	            ELSE // error not known, user have to act - leave block
	              #statInternal.diagnostics.status := #ERR_DATALOG_OPEN;
	              #statInternal.diagnostics.subfunctionStatus := #instDataLogOpen.STATUS;
	              #statInternal.diagnostics.stateNumber := #FB_STATE_DL_OPEN;
	              #statInternal.errorUserCleared := TRUE;
	            END_IF;
	            // reset instance
	            #instDataLogOpen(REQ := FALSE);
	          END_IF;
	        END_REGION DataLog open

	      #FB_STATE_DL_CREATE:
	        REGION DataLog create
	          #instDataLogCreate(REQ       := TRUE,
	                             RECORDS   := #statDataLogCommands.noOfRecords,
	                             TIMESTAMP := #statDataLogCommands.timestampFormat,
	                             NAME      := #statDataLogCommands.name,
	                             ID        := #statDataLogCommands.id,
	                             HEADER    := #statDataLogCommands.header,
	                             DATA      := #data);

	          // check if creating and opening DL is done successfully - goto write
	          IF #instDataLogCreate.DONE THEN
	            IF (#statDataLogCommands.isLoggingByInterval = TRUE) THEN
	              #statMainState := #FB_STATE_DL_WRITE;
	            ELSE // is logging by trigger
	              #statMainState := #FB_STATE_DL_WAIT_FOR_TRIGGER;
	            END_IF;
	            // reset instance
	            #instDataLogCreate(REQ := FALSE);

	            // check if error occurred
	          ELSIF #instDataLogCreate.ERROR THEN
	            // error not known, user have to act
	            #statInternal.diagnostics.status := #ERR_DATALOG_CREATE;
	            #statInternal.diagnostics.subfunctionStatus := #instDataLogCreate.STATUS;
	            #statInternal.diagnostics.stateNumber := #FB_STATE_DL_OPEN;
	            #statInternal.errorUserCleared := TRUE;
	            // reset instance
	            #instDataLogCreate(REQ := FALSE);
	          END_IF;
	        END_REGION DataLog create

	      #FB_STATE_DL_WAIT_FOR_TRIGGER,
	      #FB_STATE_DL_WAIT_FOR_WRITE_CYCLE:
	        REGION Wait for trigger
	          // reset flags
	          #statLlastEntryReached := FALSE;
	          #statInternal.diagnostics.status := #STATUS_SUBSEQUENT_CALL;

	          IF TRUE // if trigger has a rising edge
	            AND (#triggerLogEntry AND NOT #statDataLogCommands.edgeOnTriggerLogEntry)
	            AND (#statMainState = #FB_STATE_DL_WAIT_FOR_TRIGGER)
	          THEN
	            #statMainState := #FB_STATE_DL_WRITE;

	          ELSIF TRUE // if interval is over
	            AND #instIntervalTimer.Q
	            AND (#statMainState = #FB_STATE_DL_WAIT_FOR_WRITE_CYCLE)
	          THEN
	            #statMainState := #FB_STATE_DL_WRITE;
	          END_IF;
	        END_REGION Wait for trigger

	      #FB_STATE_DL_WRITE:
	        REGION DataLog write
	          #instDataLogWrite(REQ := TRUE,
	                            ID  := #statDataLogCommands.id);

	          // check if datalog is at its last entry
	          IF (#instDataLogWrite.STATUS = #DATALOG_LAST_ENTRY_WRITTEN) THEN
	            // set flag
	            #statLlastEntryReached := TRUE;
	            #statInternal.diagnostics.status := #STATUS_MAX_ENTRIES_REACHED;
	            // increment counter
	            #statNoOfEntries += 1;
	            #statWriteEntryDone := TRUE;

	            // check if datalog should be overwritten or not
	            IF #statDataLogCommands.enableRingBuffer THEN
	              // is logging by interval
	              IF #statDataLogCommands.isLoggingByInterval THEN
	                #statMainState := #FB_STATE_DL_WAIT_FOR_WRITE_CYCLE;

	              ELSE // is logging by trigger
	                #statMainState := #FB_STATE_DL_WAIT_FOR_TRIGGER;
	              END_IF;

	            ELSE // do not overwrite - disable and leave block
	              #statMainState := #FB_STATE_NO_PROCESSING;
	            END_IF;
	            // reset instance
	            #instDataLogWrite(REQ := FALSE);
	            #tempExitStateLoop := FALSE;

	            // check if open DL is done successfully - goto write
	          ELSIF #instDataLogWrite.DONE THEN
	            // increment counter
	            #statNoOfEntries += 1;
	            #statWriteEntryDone := TRUE;

	            IF #statDataLogCommands.isLoggingByInterval = TRUE THEN
	              #statMainState := #FB_STATE_DL_WAIT_FOR_WRITE_CYCLE;
	            ELSE // is logging by trigger
	              #statMainState := #FB_STATE_DL_WAIT_FOR_TRIGGER;
	            END_IF;
	            // reset instance
	            #instDataLogWrite(REQ := FALSE);
	            #tempExitStateLoop := FALSE;

	            // check if error occurred
	          ELSIF #instDataLogWrite.ERROR THEN
	            // error not known, user have to act
	            #statInternal.diagnostics.status := #ERR_DATALOG_WRITE;
	            #statInternal.diagnostics.subfunctionStatus := #instDataLogWrite.STATUS;
	            #statInternal.diagnostics.stateNumber := #FB_STATE_DL_WRITE;
	            #statInternal.errorAutoCleared := TRUE;
	            #statMainState := #FB_STATE_NO_PROCESSING;
	            // reset instance
	            #instDataLogWrite(REQ := FALSE);
	          END_IF;
	        END_REGION DataLog write

	      #FB_STATE_DL_CLEAR:
	        REGION DataLog clear
	          #instDataLogClear(REQ := TRUE,
	                            ID  := #statDataLogCommands.id);

	          // check if open DL is done successfully - goto write
	          IF #instDataLogClear.DONE THEN
	            #statMainState := #FB_STATE_DL_CLEAR_DONE;
	            // reset flag
	            #statLlastEntryReached := FALSE;
	            #statNoOfEntries := 0;
	            // reset instance
	            #instDataLogClear(REQ := FALSE);

	            // check if error occurred
	          ELSIF #instDataLogClear.ERROR THEN
	            // error not known, user have to act
	            #statInternal.diagnostics.status := #ERR_DATALOG_CLEAR;
	            #statInternal.diagnostics.subfunctionStatus := #instDataLogClear.STATUS;
	            #statInternal.diagnostics.stateNumber := #FB_STATE_DL_CLEAR;
	            #statInternal.errorAutoCleared := TRUE;
	            #statMainState := #FB_STATE_NO_PROCESSING;
	            // reset instance
	            #instDataLogWrite(REQ := FALSE);
	          END_IF;
	        END_REGION DataLog clear

	      #FB_STATE_DL_CLEAR_DONE:
	        REGION DataLog clear done
	          IF NOT #clearLog THEN
	            IF #statDataLogCommands.isLoggingByInterval THEN
	              #statMainState := #FB_STATE_DL_WRITE;
	            ELSE
	              #statMainState := #FB_STATE_DL_WAIT_FOR_TRIGGER;
	            END_IF;
	          END_IF;
	        END_REGION DataLog clear

	      #FB_STATE_DL_DELETE:
	        REGION DataLog delete
	          #instDataLogDelete(REQ     := TRUE,
	                             NAME    := #statDataLogCommands.name,
	                             DelFile := #parameter.deleteFile,
	                             ID      := #statDataLogCommands.id);

	          // check if delete DL is done successfully - goto disable completed
	          IF #instDataLogDelete.DONE THEN
	            #statMainState := #FB_STATE_DL_DELETE_DONE;
	            // reset flag
	            #statLlastEntryReached := FALSE;
	            #statNoOfEntries := 0;
	            // reset instance
	            #instDataLogDelete(REQ := FALSE);

	            // check if error occurred
	          ELSIF #instDataLogDelete.ERROR THEN
	            // error not known, user have to act
	            #statInternal.diagnostics.status := #ERR_DATALOG_DELETE;
	            #statInternal.diagnostics.subfunctionStatus := #instDataLogDelete.STATUS;
	            #statInternal.diagnostics.stateNumber := #FB_STATE_DL_DELETE;
	            #statInternal.errorAutoCleared := TRUE;
	            #statMainState := #FB_STATE_NO_PROCESSING;
	            // reset instance
	            #instDataLogDelete(REQ := FALSE);
	          END_IF;
	        END_REGION DataLog delete

	      #FB_STATE_DL_DELETE_DONE:
	        REGION DataLog delete done
	          IF NOT #deleteLog THEN
	            #statMainState := #FB_STATE_DISABLING_COMPLETED;
	          END_IF;
	        END_REGION DataLog delete

	      #FB_STATE_DISABLING: // Disabling active
	        REGION Disabling
	          // closing DataLog
	          #instDataLogClose(REQ := TRUE,
	                            ID  := #statDataLogCommands.id);

	          // check if datalog is closed
	          IF FALSE
	            OR #instDataLogClose.DONE
	            OR #instDataLogClose.STATUS = #SUB_ERR_DATALOG_DOSE_NOT_EXIST
	          THEN
	            #statMainState := #FB_STATE_DISABLING_COMPLETED;
	            #statInternal.diagnostics.status := #STATUS_FINISHED_NO_ERROR;

	            // if closing ends with error - report this as well
	          ELSIF #instDataLogClose.ERROR THEN
	            // error occurred - copy to outputs
	            #statInternal.diagnostics.status := #ERR_DATALOG_CLOSE;
	            #statInternal.diagnostics.subfunctionStatus := #instDataLogClose.STATUS;
	            #statInternal.diagnostics.stateNumber := #FB_STATE_DISABLING;
	            #statInternal.errorAutoCleared := TRUE;// next state
	            #statMainState := #FB_STATE_DISABLING_COMPLETED;
	          END_IF;
	        END_REGION Disabling

	      #FB_STATE_DISABLING_COMPLETED:
	        REGION Disabling completed
	          // reset instance
	          #instDataLogClose(REQ := FALSE);
	          // When disabling is complete the bit #statDisablingCompleted must be set
	          #statInternal.disablingCompleted := TRUE;
	        END_REGION Disabling completed

	      ELSE // Undefined state in state machine reached
	        REGION Undefined state
	          #statInternal.diagnostics.status := #ERR_UNDEFINED_STATE;
	          #statInternal.diagnostics.subfunctionStatus := #SUB_STATUS_NO_ERROR;
	          #statInternal.diagnostics.stateNumber := #statMainState;
	          #statInternal.errorUserCleared := TRUE;
	        END_REGION Undefined state
	    END_CASE;

	    // call interval timer
	    #instIntervalTimer.TON(IN := (#statMainState = #FB_STATE_DL_WAIT_FOR_WRITE_CYCLE),
	                           PT := #statDataLogCommands.loggingInterval);    // if one ore more runs in the same cycle are necessary, set #tempExitStateLoop := FALSE;
	    // check state, if condition = TRUE --> #tempExitStateLoop = TRUE --> LEAVE LOOP
	  UNTIL (TRUE = #tempExitStateLoop)
	  END_REPEAT;
	END_REGION STATE_MACHINE

	REGION Edge memory
	  // store/ reset edge memory
	  #statDataLogCommands.edgeOnTriggerLogEntry := #triggerLogEntry;
	  #statDataLogCommands.clearLogPrevious := #clearLog;
	  #statDataLogCommands.deleteLogPrevious := #deleteLog;
	END_REGION

	REGION OUTPUTS
	  // Write outputs
	  IF (#statInternal.disablingCompleted = TRUE) THEN
	    REGION disabling
	      // Reset outputs if disabling completed
	      #statInternal.valid := FALSE;
	      #statInternal.busy := FALSE;
	      #statInternal.error := FALSE;
	      #statInternal.errorUserCleared := FALSE;
	      #statInternal.errorAutoCleared := FALSE;
	      #statInternal.diagnostics.status := #STATUS_NO_CALL;
	      // Reset application specific outputs
	      #statWriteEntryDone := FALSE;
	    END_REGION disabling

	  ELSIF (#statInternal.errorUserCleared = TRUE) AND (#statInternal.error = FALSE) THEN
	    REGION error user cleared
	      // Error can only be cleared by user; rising edge at enable input is needed to continue
	      #statInternal.valid := FALSE;
	      #statInternal.busy := FALSE;
	      #statInternal.error := TRUE;
	      // Write diagnostics
	      #diagnostics := #statInternal.diagnostics;
	      // Reset application specific outputs
	      #statWriteEntryDone := FALSE;
	      // execution aborted --> set state no processing
	      #statMainState := #FB_STATE_NO_PROCESSING;
	    END_REGION error user cleared

	  ELSIF (#statInternal.errorAutoCleared = TRUE) AND (#statInternal.error = FALSE) THEN
	    REGION error auto cleared
	      // Error can be reset by FB automatically
	      #statInternal.valid := FALSE;
	      #statInternal.busy := TRUE;
	      #statInternal.error := TRUE;
	      // Write diagnostics
	      #diagnostics := #statInternal.diagnostics;
	      // Reset application specific outputs
	      #statWriteEntryDone := FALSE;
	    END_REGION error auto cleared

	  ELSIF (#statInternal.errorAutoCleared = FALSE) AND (#statInternal.errorUserCleared = FALSE) AND (#statInternal.error = TRUE) THEN
	    REGION after user/auto cleared
	      // If autocleared error is acknowledged
	      #statInternal.valid := TRUE;
	      #statInternal.busy := TRUE;
	      #statInternal.error := FALSE;
	      // remove this line if more detailed status information is used instead of "#STATUS_SUBSEQUENT_CALL"
	      #statInternal.diagnostics.status := #STATUS_SUBSEQUENT_CALL;
	    END_REGION after user/auto cleared
	  END_IF;

	  REGION Write static values to outputs
	    #valid := #statInternal.valid;
	    #busy := #statInternal.busy;
	    #error := #statInternal.error;
	    #status := #statInternal.diagnostics.status;
	    // if ENO mechanism is not used / not wanted replace the following line by --> ENO := TRUE;
	    ENO := NOT #statInternal.error;
	    // Write application specific static values to outputs
	    #lastEntryReached := #statLlastEntryReached;
	    #noOfEntries := #statNoOfEntries;

	    #writeEntryDone := #statWriteEntryDone;
	    #statWriteEntryDone := FALSE;

	    #clearLogDone := #statMainState = #FB_STATE_DL_CLEAR_DONE;
	    #deleteLogDone := #statMainState = #FB_STATE_DL_DELETE_DONE;
	  END_REGION Write static values to outputs
	END_REGION OUTPUTS

END_FUNCTION_BLOCK

FUNCTION "LGF_IsParityOdd" : Bool
{ S7_Optimized_Access := 'TRUE' }
AUTHOR : Siemens_SIMATIC_Systems_Support
FAMILY : LGF
NAME : LGF_IsParityOdd
   VAR_INPUT
      doubleWord : DWord;
   END_VAR

   VAR_TEMP
      tempDword : DWord;
   END_VAR

   VAR CONSTANT
      SHIFT_ONE_BIT : USInt := 1;
      SHIFT_TWO_BIT : USInt := 2;
      SHIFT_TO_RESULT : USInt := 28;
      MASK_FOR_RESULT : DWord := 16#11111111;
   END_VAR


BEGIN
	REGION Block info header
	  //============================================================================
	  // SIEMENS AG / (c)Copyright 2018
	  //----------------------------------------------------------------------------
	  // Title:            LGF_IsParityOdd
	  // Comment/Function: check if parity in input tag is odd
	  //                   if number of bits is odd, return TRUE
	  //                   https://graphics.stanford.edu/~seander/bithacks.html#ParityMultiply
	  //                   ENO not needed, no error possible
	  // Library/Family:   LGF (Library General Functions)
	  // Author:           Siemens Digital Industry Support
	  // Tested with:      S7-PLCSIM Advanced V2.0 SP1
	  // Engineering:      TIA Portal V15 Update 2
	  // Restrictions:     ENO not needed, no error possible
	  // Requirements:     PLC (S7-1200 / S7-1500)
	  //-------------------------------------------------------------------------------
	  // Change log table:
	  // Version  | Date       | Expert in charge       | Changes applied
	  //----------|------------|------------------------|------------------------------
	  // 01.00.00 | 2019.11.28 | Simatic Systems Support
	  //                         First released version
	  // 03.00.00 | 23.04.2020 | Simatic Systems Support | Set version to V3.0.0
	  //                         harmonize the version of the whole library
	  // 03.00.01 | 12.11.2020 | Simatic Systems Support
	  //                         Insert documentation
	  //=============================================================================
	END_REGION Block info header

	REGION DESCRIPTION
	  (/**/)
	END_REGION DESCRIPTION

	REGION Logic
	  #tempDword := #doubleWord; // 32-bit word
	  #tempDword := #tempDword XOR SHR(IN := #tempDword, N := #SHIFT_ONE_BIT);
	  #tempDword := #tempDword XOR SHR(IN := #tempDword, N := #SHIFT_TWO_BIT);

	  #tempDword := UDINT_TO_DWORD(DWORD_TO_UDINT(#tempDword AND #MASK_FOR_RESULT) * DWORD_TO_UDINT(#MASK_FOR_RESULT));

	  #tempDword := SHR(IN := #tempDword, N := #SHIFT_TO_RESULT);

	  // result is stored in LSB
	  #LGF_IsParityOdd := #tempDword.%X0;

	  // eno not needed, no error possible
	  ENO := FALSE;
	END_REGION

END_FUNCTION

FUNCTION "LGF_CalcCRC32Advanced" : DWord
{ S7_Optimized_Access := 'TRUE' }
AUTHOR : Siemens_Industry_Support
FAMILY : LGF
NAME : LGF_CRC32Advanced
   VAR_INPUT
      initValue { S7_PredefinedAssignment := '16#00'} : DWord;
      mask { S7_PredefinedAssignment := '16#00'} : DWord;
      finalXorValue { S7_PredefinedAssignment := '16#00'} : DWord;
      reflectInput { S7_PredefinedAssignment := 'FALSE'} : Bool;
      reflectResult { S7_PredefinedAssignment := 'FALSE'} : Bool;
      noOfElements { S7_PredefinedAssignment := '0'} : UInt;
   END_VAR

   VAR_OUTPUT
      error : Bool;
      status : Word;
   END_VAR

   VAR_IN_OUT
      "array" : Array[*] of Byte;
   END_VAR

   VAR_TEMP
      tempInput : Byte;
      tempCRC : DWord;
      tempInvCRC : DWord;
      tempLowerLimit : DInt;
      tempUpperLimit : DInt;
      tempIndexArray : DInt;
      tempIndexCRC : DInt;
   END_VAR

   VAR CONSTANT
      SHIFT_ONE_BIT : UInt := 1;
      SHIFT_THREE_BYTE : UInt := 24;
      ARRAY_FIRST_DIMENSION : UInt := 1;
      CRC_LOOP_LOWER_LIMIT : DInt := 0;
      CRC_LOOP_UPPER_LIMIT : DInt := 7;
      STATUS_NO_ERROR : Word := 16#0000;
      ERR_NO_OF_ELEMENTS : Word := 16#8400;
   END_VAR


BEGIN
	REGION Block info header
	  //===============================================================================
	  // SIEMENS AG / (c)Copyright 2019
	  //-------------------------------------------------------------------------------
	  // Title:            LGF_CRC32Advanced
	  // Comment/Function: This function makes a CRC calculation according
	  //                   to the CRC-32 algorithm
	  //                   advanced because of reflect In/Out and final XOR combination
	  // Library/Family:   LGF (Library General Functions)
	  // Author:           Siemens Digital Industry Support
	  // Tested with:      CPU 1515F-2 PN FW:V2.6
	  // Engineering:      TIA Portal V15.1 Update 2
	  // Restrictions:     ENO disabled - no error handling, no failure possible
	  // Requirements:     PLC (S7-1200 / S7-1500)
	  //-------------------------------------------------------------------------------
	  // Change log table:
	  // Version  | Date       | Expert in charge       | Changes applied
	  //----------|------------|------------------------|------------------------------
	  // 01.00.00 03.07.2018  Siemens Industry Online Support
	  //                      First released version
	  // 01.00.01 17.08.2018  Siemens Industry Online Support
	  //                      Upgrade: TIA V15 Update 2
	  // 01.00.02 23.11.2018  Siemens Industry Online Support
	  //                      Upgrade: TIA V15.1
	  // 01.00.03 09.10.2019  Simatic Systems Support
	  //                      Code refactoring, comments added
	  // 03.00.00 23.04.2020  Simatic Systems Support
	  //                      Set version to V3.0.0, harmonize the version of the whole library
	  // 03.00.01 12.11.2020  Simatic Systems Support
	  //                      Insert documentation
	  //                      Assign default start values to optional inputs - `initValue`, `mask`, `finalXorValue`, `reflectInput`, `reflectResult`
	  // 03.01.00 14.04.2023  Simatic Systems Support
	  //                      Add input `noOfElements` to assign length to be converted different from array size
	  //                      Add outputs `error` and `status` display a wrong assignment to `noOfElements`
	  //=============================================================================
	END_REGION Block info header

	REGION DESCRIPTION
	  (/**/)
	END_REGION DESCRIPTION

	REGION Initialization and input data processing
	  // Defining initial value for algorithm
	  #tempCRC := #initValue;
	  // Input array size calculation
	  #tempLowerLimit := LOWER_BOUND(ARR := #array, DIM := #ARRAY_FIRST_DIMENSION);
	  #tempUpperLimit := UPPER_BOUND(ARR := #array, DIM := #ARRAY_FIRST_DIMENSION);

	  // check paramter `noOfELements`, if gretaer than zero check if fits to array size
	  IF #noOfElements > 0 THEN
	    IF #noOfElements > (#tempUpperLimit - #tempLowerLimit + 1) THEN
	      #status := #ERR_NO_OF_ELEMENTS;
	      #error := TRUE;
	      ENO := FALSE;
	      #LGF_CalcCRC32Advanced := #tempCRC;
	      RETURN;
	    ELSE
	      #tempUpperLimit := #tempLowerLimit + #noOfElements - 1;
	    END_IF;
	  END_IF;
	END_REGION

	REGION CRC calculation
	  FOR #tempIndexArray := #tempLowerLimit TO #tempUpperLimit DO

	    IF #reflectInput THEN
	      // Reverse bit order in input byte
	      #tempInput.%X7 := #array[#tempIndexArray].%X0;
	      #tempInput.%X6 := #array[#tempIndexArray].%X1;
	      #tempInput.%X5 := #array[#tempIndexArray].%X2;
	      #tempInput.%X4 := #array[#tempIndexArray].%X3;
	      #tempInput.%X3 := #array[#tempIndexArray].%X4;
	      #tempInput.%X2 := #array[#tempIndexArray].%X5;
	      #tempInput.%X1 := #array[#tempIndexArray].%X6;
	      #tempInput.%X0 := #array[#tempIndexArray].%X7;
	    ELSE
	      #tempInput := #array[#tempIndexArray];
	    END_IF;

	    // Perform division using XOR function for appropriate DWord in array (with shift byte into MSB of 32bit CRC)
	    #tempCRC := #tempCRC XOR SHL(IN := BYTE_TO_DWORD(#tempInput), N := #SHIFT_THREE_BYTE);

	    FOR #tempIndexCRC := #CRC_LOOP_LOWER_LIMIT TO #CRC_LOOP_UPPER_LIMIT DO
	      // Check if MSB is set
	      IF #tempCRC.%X31 THEN
	        // Shift left and perform division by mask polynomial using XOR function
	        #tempCRC := SHL(IN := #tempCRC, N := #SHIFT_ONE_BIT) XOR #mask;
	      ELSE
	        // Shift left without division
	        #tempCRC := SHL(IN := #tempCRC, N := #SHIFT_ONE_BIT);
	      END_IF;
	    END_FOR;

	  END_FOR;
	END_REGION

	REGION Outputs assignment
	  IF #reflectResult THEN
	    // Reverse bit order in CRC checksum
	    #tempInvCRC.%X31 := #tempCRC.%X0;
	    #tempInvCRC.%X30 := #tempCRC.%X1;
	    #tempInvCRC.%X29 := #tempCRC.%X2;
	    #tempInvCRC.%X28 := #tempCRC.%X3;
	    #tempInvCRC.%X27 := #tempCRC.%X4;
	    #tempInvCRC.%X26 := #tempCRC.%X5;
	    #tempInvCRC.%X25 := #tempCRC.%X6;
	    #tempInvCRC.%X24 := #tempCRC.%X7;
	    #tempInvCRC.%X23 := #tempCRC.%X8;
	    #tempInvCRC.%X22 := #tempCRC.%X9;
	    #tempInvCRC.%X21 := #tempCRC.%X10;
	    #tempInvCRC.%X20 := #tempCRC.%X11;
	    #tempInvCRC.%X19 := #tempCRC.%X12;
	    #tempInvCRC.%X18 := #tempCRC.%X13;
	    #tempInvCRC.%X17 := #tempCRC.%X14;
	    #tempInvCRC.%X16 := #tempCRC.%X15;
	    #tempInvCRC.%X15 := #tempCRC.%X16;
	    #tempInvCRC.%X14 := #tempCRC.%X17;
	    #tempInvCRC.%X13 := #tempCRC.%X18;
	    #tempInvCRC.%X12 := #tempCRC.%X19;
	    #tempInvCRC.%X11 := #tempCRC.%X20;
	    #tempInvCRC.%X10 := #tempCRC.%X21;
	    #tempInvCRC.%X9 := #tempCRC.%X22;
	    #tempInvCRC.%X8 := #tempCRC.%X23;
	    #tempInvCRC.%X7 := #tempCRC.%X24;
	    #tempInvCRC.%X6 := #tempCRC.%X25;
	    #tempInvCRC.%X5 := #tempCRC.%X26;
	    #tempInvCRC.%X4 := #tempCRC.%X27;
	    #tempInvCRC.%X3 := #tempCRC.%X28;
	    #tempInvCRC.%X2 := #tempCRC.%X29;
	    #tempInvCRC.%X1 := #tempCRC.%X30;
	    #tempInvCRC.%X0 := #tempCRC.%X31;

	    #LGF_CalcCRC32Advanced := #tempInvCRC XOR #finalXorValue;
	  ELSE
	    #LGF_CalcCRC32Advanced := #tempCRC XOR #finalXorValue;
	  END_IF;

	  #status := #STATUS_NO_ERROR;
	  #error := FALSE;
	  ENO := TRUE;
	END_REGION

END_FUNCTION

FUNCTION "LGF_CalcCRC32" : DWord
{ S7_Optimized_Access := 'TRUE' }
AUTHOR : Siemens_Industry_Support
FAMILY : LGF
NAME : LGF_CRC32
   VAR_INPUT
      initValue { S7_PredefinedAssignment := '16#00'} : DWord;
      mask { S7_PredefinedAssignment := '16#00'} : DWord;
      noOfElements { S7_PredefinedAssignment := '0'} : UInt;
   END_VAR

   VAR_OUTPUT
      error : Bool;
      status : Word;
   END_VAR

   VAR_IN_OUT
      "array" : Array[*] of Byte;
   END_VAR

   VAR_TEMP
      tempCRC : DWord;
      tempLowerLimit : DInt;
      tempUpperLimit : DInt;
      tempIndexArray : DInt;
      tempIndexCRC : DInt;
   END_VAR

   VAR CONSTANT
      SHIFT_ONE_BIT : UInt := 1;
      SHIFT_THREE_BYTES : UInt := 24;
      ARRAY_FIRST_DIMENSION : UInt := 1;
      CRC_LOOP_LOWER_LIMIT : DInt := 0;
      CRC_LOOP_UPPER_LIMIT : DInt := 7;
      STATUS_NO_ERROR : Word := 16#0000;
      ERR_NO_OF_ELEMENTS : Word := 16#8400;
   END_VAR


BEGIN
	REGION Block info header
	  //===============================================================================
	  // SIEMENS AG / (c)Copyright 2019
	  //-------------------------------------------------------------------------------
	  // Title:            LGF_CRC32
	  // Comment/Function: This function makes a CRC calculation according
	  //                   to the CRC-32 algorithm
	  // Library/Family:   LGF (Library General Functions)
	  // Author:           Siemens Digital Industry Support
	  // Tested with:      CPU 1515F-2 PN FW:V2.6
	  // Engineering:      TIA Portal V15.1 Update 2
	  // Restrictions:     ENO disabled - no error handling, no failure possible
	  // Requirements:     PLC (S7-1200 / S7-1500)
	  //-------------------------------------------------------------------------------
	  // Change log table:
	  // Version  | Date       | Expert in charge       | Changes applied
	  //----------|------------|------------------------|------------------------------
	  // 01.00.00 03.07.2018  Siemens Industry Online Support
	  //                      First released version
	  // 01.00.01 17.08.2018  Siemens Industry Online Support
	  //                      Upgrade: TIA V15 Update 2
	  // 01.00.02 23.11.2018  Siemens Industry Online Support
	  //                      Upgrade: TIA V15.1
	  // 01.00.03 09.10.2019  Simatic Systems Support
	  //                      Code refactoring, comments added
	  // 03.00.00 23.04.2020  Simatic Systems Support
	  //                      Set version to V3.0.0, harmonize the version of the whole library
	  // 03.00.01 12.11.2020  Simatic Systems Support
	  //                      Insert documentation
	  //                      Assign default start values to optional inputs - `initValue`, `mask`
	  // 03.01.00 14.04.2023  Simatic Systems Support
	  //                      Add input `noOfElements` to assign length to be converted different from array size
	  //                      Add outputs `error` and `status` display a wrong assignment to `noOfElements`
	  //=============================================================================
	END_REGION Block info header

	REGION DESCRIPTION
	  (/**/)
	END_REGION DESCRIPTION

	REGION Initialization and input data processing
	  // Defining initial value for algorithm
	  #tempCRC := #initValue;
	  // Input array size calculation
	  #tempLowerLimit := LOWER_BOUND(ARR := #array, DIM := #ARRAY_FIRST_DIMENSION);
	  #tempUpperLimit := UPPER_BOUND(ARR := #array, DIM := #ARRAY_FIRST_DIMENSION);

	  // check paramter `noOfELements`, if gretaer than zero check if fits to array size
	  IF #noOfElements > 0 THEN
	    IF #noOfElements > (#tempUpperLimit - #tempLowerLimit + 1) THEN
	      #status := #ERR_NO_OF_ELEMENTS;
	      #error := TRUE;
	      ENO := FALSE;
	      #LGF_CalcCRC32 := #tempCRC;
	      RETURN;
	    ELSE
	      #tempUpperLimit := #tempLowerLimit + #noOfElements - 1;
	    END_IF;
	  END_IF;
	END_REGION

	REGION CRC calculation
	  FOR #tempIndexArray := #tempLowerLimit TO #tempUpperLimit DO
	    // Perform division using XOR function for appropriate word in array (with shift byte into MSB of 32bit CRC)
	    #tempCRC := #tempCRC XOR SHL(IN := BYTE_TO_DWORD(#array[#tempIndexArray]), N := #SHIFT_THREE_BYTES);

	    FOR #tempIndexCRC := #CRC_LOOP_LOWER_LIMIT TO #CRC_LOOP_UPPER_LIMIT DO
	      // Check if MSB is set
	      IF #tempCRC.%X31 THEN
	        // Shift left and perform division by mask polynomial using XOR function
	        #tempCRC := SHL(IN := #tempCRC, N := #SHIFT_ONE_BIT) XOR #mask;
	      ELSE
	        // Shift left without division
	        #tempCRC := SHL(IN := #tempCRC, N := #SHIFT_ONE_BIT);
	      END_IF;
	    END_FOR;

	  END_FOR;
	END_REGION

	REGION Outputs assignment
	  #LGF_CalcCRC32 := #tempCRC;

	  #status := #STATUS_NO_ERROR;
	  #error := FALSE;
	  ENO := TRUE;
	END_REGION

END_FUNCTION

FUNCTION "LGF_CalcCRC16Advanced" : Word
{ S7_Optimized_Access := 'TRUE' }
AUTHOR : Siemens_Industry_Support
FAMILY : LGF
NAME : LGF_CRC16Advanced
   VAR_INPUT
      initValue { S7_PredefinedAssignment := '16#00'} : Word;
      mask { S7_PredefinedAssignment := '16#00'} : Word;
      finalXorValue { S7_PredefinedAssignment := '16#00'} : Word;
      reflectInput { S7_PredefinedAssignment := 'FALSE'} : Bool;
      reflectResult { S7_PredefinedAssignment := 'FALSE'} : Bool;
      noOfElements { S7_PredefinedAssignment := '0'} : UInt;
   END_VAR

   VAR_OUTPUT
      error : Bool;
      status : Word;
   END_VAR

   VAR_IN_OUT
      "array" : Array[*] of Byte;
   END_VAR

   VAR_TEMP
      tempInput : Byte;
      tempCRC : Word;
      tempInvCRC : Word;
      tempLowerLimit : DInt;
      tempUpperLimit : DInt;
      tempIndexArray : DInt;
      tempIndexCRC : DInt;
   END_VAR

   VAR CONSTANT
      SHIFT_ONE_BIT : UInt := 1;
      SHIFT_ONE_BYTE : UInt := 8;
      ARRAY_FIRST_DIMENSION : UInt := 1;
      CRC_LOOP_LOWER_LIMIT : DInt := 0;
      CRC_LOOP_UPPER_LIMIT : DInt := 7;
      STATUS_NO_ERROR : Word := 16#0000;
      ERR_NO_OF_ELEMENTS : Word := 16#8400;
   END_VAR


BEGIN
	REGION Block info header
	  //===============================================================================
	  // SIEMENS AG / (c)Copyright 2019
	  //-------------------------------------------------------------------------------
	  // Title:            LGF_CRC16Advanced
	  // Comment/Function: This function makes a CRC calculation according
	  //                   to the CRC-16 advanced algorithm
	  //                   advanced because of reflect In/Out and final XOR combination
	  // Library/Family:   LGF (Library General Functions)
	  // Author:           Siemens Digital Industry Support
	  // Tested with:      CPU 1515F-2 PN FW:V2.6
	  // Engineering:      TIA Portal V15.1 Update 2
	  // Restrictions:     ENO disabled - no error handling, no failure possible
	  // Requirements:     PLC (S7-1200 / S7-1500)
	  //-------------------------------------------------------------------------------
	  // Change log table:
	  // Version  | Date       | Expert in charge       | Changes applied
	  //----------|------------|------------------------|------------------------------
	  // 01.00.00 16.12.2019  Simatic Systems Support
	  //                      first release, copied from "LGF_CalcCRC32Advanced"
	  // 03.00.00 23.04.2020  Simatic Systems Support
	  //                      Set version to V3.0.0, harmonize the version of the whole library
	  // 03.00.01 12.11.2020  Simatic Systems Support
	  //                      Insert documentation
	  //                      Assign default start values to optional inputs - `initValue`, `mask`, `finalXorValue`, `reflectInput`, `reflectResult`
	  // 03.01.00 14.04.2023  Simatic Systems Support
	  //                      Add input `noOfElements` to assign length to be converted different from array size
	  //                      Add outputs `error` and `status` display a wrong assignment to `noOfElements`
	  //=============================================================================
	END_REGION Block info header

	REGION DESCRIPTION
	  (/**/)
	END_REGION DESCRIPTION

	REGION Initialization and input data processing
	  // Defining initial value for algorithm
	  #tempCRC := #initValue;
	  // Input array size calculation
	  #tempLowerLimit := LOWER_BOUND(ARR := #array, DIM := #ARRAY_FIRST_DIMENSION);
	  #tempUpperLimit := UPPER_BOUND(ARR := #array, DIM := #ARRAY_FIRST_DIMENSION);

	  // check paramter `noOfELements`, if gretaer than zero check if fits to array size
	  IF #noOfElements > 0 THEN
	    IF #noOfElements > (#tempUpperLimit - #tempLowerLimit + 1) THEN
	      #status := #ERR_NO_OF_ELEMENTS;
	      #error := TRUE;
	      ENO := FALSE;
	      #LGF_CalcCRC16Advanced := #tempCRC;
	      RETURN;
	    ELSE
	      #tempUpperLimit := #tempLowerLimit + #noOfElements - 1;
	    END_IF;
	  END_IF;
	END_REGION

	REGION CRC calculation
	  FOR #tempIndexArray := #tempLowerLimit TO #tempUpperLimit DO

	    IF #reflectInput THEN
	      // Reverse bit order in input byte
	      #tempInput.%X7 := #array[#tempIndexArray].%X0;
	      #tempInput.%X6 := #array[#tempIndexArray].%X1;
	      #tempInput.%X5 := #array[#tempIndexArray].%X2;
	      #tempInput.%X4 := #array[#tempIndexArray].%X3;
	      #tempInput.%X3 := #array[#tempIndexArray].%X4;
	      #tempInput.%X2 := #array[#tempIndexArray].%X5;
	      #tempInput.%X1 := #array[#tempIndexArray].%X6;
	      #tempInput.%X0 := #array[#tempIndexArray].%X7;
	    ELSE
	      #tempInput := #array[#tempIndexArray];
	    END_IF;

	    // Perform division using XOR function for appropriate Word in array (with shift byte into MSB of 16bit CRC)
	    #tempCRC := #tempCRC XOR SHL(IN := BYTE_TO_WORD(#tempInput), N := #SHIFT_ONE_BYTE);

	    FOR #tempIndexCRC := #CRC_LOOP_LOWER_LIMIT TO #CRC_LOOP_UPPER_LIMIT DO
	      // Check if MSB is set
	      IF #tempCRC.%X15 THEN
	        // Shift left and perform division by mask polynomial using XOR function
	        #tempCRC := SHL(IN := #tempCRC, N := #SHIFT_ONE_BIT) XOR #mask;
	      ELSE
	        // Shift left without division
	        #tempCRC := SHL(IN := #tempCRC, N := #SHIFT_ONE_BIT);
	      END_IF;
	    END_FOR;

	  END_FOR;
	END_REGION

	REGION Outputs assignment
	  IF #reflectResult THEN
	    // Reverse bit order in CRC checksum
	    #tempInvCRC.%X15 := #tempCRC.%X0;
	    #tempInvCRC.%X14 := #tempCRC.%X1;
	    #tempInvCRC.%X13 := #tempCRC.%X2;
	    #tempInvCRC.%X12 := #tempCRC.%X3;
	    #tempInvCRC.%X11 := #tempCRC.%X4;
	    #tempInvCRC.%X10 := #tempCRC.%X5;
	    #tempInvCRC.%X9 := #tempCRC.%X6;
	    #tempInvCRC.%X8 := #tempCRC.%X7;
	    #tempInvCRC.%X7 := #tempCRC.%X8;
	    #tempInvCRC.%X6 := #tempCRC.%X9;
	    #tempInvCRC.%X5 := #tempCRC.%X10;
	    #tempInvCRC.%X4 := #tempCRC.%X11;
	    #tempInvCRC.%X3 := #tempCRC.%X12;
	    #tempInvCRC.%X2 := #tempCRC.%X13;
	    #tempInvCRC.%X1 := #tempCRC.%X14;
	    #tempInvCRC.%X0 := #tempCRC.%X15;

	    #LGF_CalcCRC16Advanced := #tempInvCRC XOR #finalXorValue;
	  ELSE
	    #LGF_CalcCRC16Advanced := #tempCRC XOR #finalXorValue;
	  END_IF;

	  #status := #STATUS_NO_ERROR;
	  #error := FALSE;
	  ENO := TRUE;
	END_REGION

END_FUNCTION

FUNCTION "LGF_CalcCRC16" : Word
{ S7_Optimized_Access := 'TRUE' }
AUTHOR : Siemens_Industry_Support
FAMILY : LGF
NAME : LGF_CRC16
   VAR_INPUT
      initValue { S7_PredefinedAssignment := '16#00'} : Word;
      mask { S7_PredefinedAssignment := '16#00'} : Word;
      noOfElements { S7_PredefinedAssignment := '0'} : UInt;
   END_VAR

   VAR_OUTPUT
      error : Bool;
      status : Word;
   END_VAR

   VAR_IN_OUT
      "array" : Array[*] of Byte;
   END_VAR

   VAR_TEMP
      tempCRC : Word;
      tempLowerLimit : DInt;
      tempUpperLimit : DInt;
      tempIndexArray : DInt;
      tempIndexCRC : DInt;
   END_VAR

   VAR CONSTANT
      SHIFT_ONE_BIT : UInt := 1;
      SHIFT_ONE_BYTE : UInt := 8;
      ARRAY_FIRST_DIMENSION : UInt := 1;
      CRC_LOOP_LOWER_LIMIT : DInt := 0;
      CRC_LOOP_UPPER_LIMIT : DInt := 7;
      ERR_NO_OF_ELEMENTS : Word := 16#8400;
      STATUS_NO_ERROR : Word := 16#0000;
   END_VAR


BEGIN
	REGION Block info header
	  //===============================================================================
	  // SIEMENS AG / (c)Copyright 2019
	  //-------------------------------------------------------------------------------
	  // Title:            LGF_CRC16
	  // Comment/Function: This function makes a CRC calculation according
	  //                   to the CRC-16 algorithm
	  // Library/Family:   LGF (Library General Functions)
	  // Author:           Siemens Digital Industry Support
	  // Tested with:      CPU 1515F-2 PN FW:V2.6
	  // Engineering:      TIA Portal V15.1 Update 2
	  // Restrictions:     ENO disabled - no error handling, no failure possible
	  // Requirements:     PLC (S7-1200 / S7-1500)
	  //-------------------------------------------------------------------------------
	  // Change log table:
	  // Version  | Date       | Expert in charge       | Changes applied
	  //----------|------------|------------------------|------------------------------
	  // 01.00.00 03.07.2018  Siemens Industry Online Support
	  //                      First released version
	  // 01.00.01 17.08.2018  Siemens Industry Online Support
	  //                      Upgrade: TIA V15 Update 2
	  // 01.00.02 23.11.2018  Siemens Industry Online Support
	  //                      Upgrade: TIA V15.1
	  // 01.00.03 09.10.2019  Simatic Systems Support
	  //                      Code refactoring, comments added
	  // 03.00.00 23.04.2020  Simatic Systems Support
	  //                      Set version to V3.0.0, harmonize the version of the whole library
	  // 03.00.01 12.11.2020  Simatic Systems Support
	  //                      Insert documentation
	  //                      Assign default start values to optional inputs - `initValue`, `mask`
	  // 03.01.00 14.04.2023  Simatic Systems Support
	  //                      Add input `noOfElements` to assign length to be converted different from array size
	  //                      Add outputs `error` and `status` display a wrong assignment to `noOfElements`
	  //=============================================================================
	END_REGION Block info header

	REGION DESCRIPTION
	  (/**/)
	END_REGION DESCRIPTION

	REGION Initialization and input data processing
	  // Defining initial value for algorithm
	  #tempCRC := #initValue;
	  // Input array size calculation
	  #tempLowerLimit := LOWER_BOUND(ARR := #array, DIM := #ARRAY_FIRST_DIMENSION);
	  #tempUpperLimit := UPPER_BOUND(ARR := #array, DIM := #ARRAY_FIRST_DIMENSION);

	  // check paramter `noOfELements`, if gretaer than zero check if fits to array size
	  IF #noOfElements > 0 THEN
	    IF #noOfElements > (#tempUpperLimit - #tempLowerLimit + 1) THEN
	      #status := #ERR_NO_OF_ELEMENTS;
	      #error := TRUE;
	      ENO := FALSE;
	      #LGF_CalcCRC16 := #tempCRC;
	      RETURN;
	    ELSE
	      #tempUpperLimit := #tempLowerLimit + #noOfElements - 1;
	    END_IF;
	  END_IF;
	END_REGION

	REGION CRC calculation
	  FOR #tempIndexArray := #tempLowerLimit TO #tempUpperLimit DO
	    // Perform division using XOR function for appropriate word in array (with shift byte into MSB of 16bit CRC)
	    #tempCRC := #tempCRC XOR SHL(IN := BYTE_TO_WORD(#array[#tempIndexArray]), N := #SHIFT_ONE_BYTE);

	    FOR #tempIndexCRC := #CRC_LOOP_LOWER_LIMIT TO #CRC_LOOP_UPPER_LIMIT DO
	      // Check if MSB is set
	      IF #tempCRC.%X15 THEN
	        // Shift left and perform division by mask polynomial using XOR function
	        #tempCRC := SHL(IN := #tempCRC, N := #SHIFT_ONE_BIT) XOR #mask;
	      ELSE
	        // Shift left without division
	        #tempCRC := SHL(IN := #tempCRC, N := #SHIFT_ONE_BIT);
	      END_IF;
	    END_FOR;

	  END_FOR;
	END_REGION

	REGION Outputs assignment
	  #LGF_CalcCRC16 := #tempCRC;

	  #status := #STATUS_NO_ERROR;
	  #error := FALSE;
	  ENO := TRUE;
	END_REGION

END_FUNCTION

FUNCTION "LGF_CalcCRC8For1Byte" : Byte
{ S7_Optimized_Access := 'TRUE' }
AUTHOR : Siemens_Industry_Support
FAMILY : LGF
NAME : LGF_CRC8For1Byte
   VAR_INPUT
      initValue { S7_PredefinedAssignment := '16#00'} : Byte;
      mask { S7_PredefinedAssignment := '16#00'} : Byte;
      value : Byte;
   END_VAR

   VAR_TEMP
      tempCRC : Byte;
      tempIndexCRC : DInt;
   END_VAR

   VAR CONSTANT
      SHIFT_ONE_BIT : UInt := 1;
      CRC_LOOP_LOWER_LIMIT : DInt := 0;
      CRC_LOOP_UPPER_LIMIT : DInt := 7;
   END_VAR


BEGIN
	REGION Block info header
	  //===============================================================================
	  // SIEMENS AG / (c)Copyright 2019
	  //-------------------------------------------------------------------------------
	  // Title:            LGF_CRC8For1Byte
	  // Comment/Function: This function makes a CRC calculation according
	  //                   to the CRC-8 algorithm for 1 byte
	  // Library/Family:   LGF (Library General Functions)
	  // Author:           Siemens Digital Industry Support
	  // Tested with:      CPU 1515F-2 PN FW:V2.6
	  // Engineering:      TIA Portal V15.1 Update 2
	  // Restrictions:     ENO disabled - no error handling, no failure possible
	  // Requirements:     PLC (S7-1200 / S7-1500)
	  //-------------------------------------------------------------------------------
	  // Change log table:
	  // Version  | Date       | Expert in charge       | Changes applied
	  //----------|------------|------------------------|------------------------------
	  // 01.00.00 03.07.2018  Siemens Industry Online Support
	  //                      First released version
	  // 01.00.01 17.08.2018  Siemens Industry Online Support
	  //                      Upgrade: TIA V15 Update 2
	  // 01.00.02 23.11.2018  Siemens Industry Online Support
	  //                      Upgrade: TIA V15.1
	  // 01.00.03 09.10.2019  Simatic Systems Support
	  //                      Code refactoring, comments added
	  // 03.00.00 23.04.2020  Simatic Systems Support
	  //                      Set version to V3.0.0, harmonize the version of the whole library
	  // 03.00.01 12.11.2020  Simatic Systems Support
	  //                      Insert documentation
	  //                      Assign default start values to optional inputs - `initValue`, `mask`
	  //=============================================================================
	END_REGION Block info header

	REGION DESCRIPTION
	  (/**/)
	END_REGION DESCRIPTION

	REGION Initialization and input data processing
	  // Defining initial value for algorithm
	  #tempCRC := #initValue XOR #value;
	END_REGION

	REGION CRC calculation
	  FOR #tempIndexCRC := #CRC_LOOP_LOWER_LIMIT TO #CRC_LOOP_UPPER_LIMIT DO
	    // Check if MSB is set
	    IF #tempCRC.%X7 THEN
	      // Shift left and perform division by mask polynomial using XOR function
	      #tempCRC := SHL(IN := #tempCRC, N := #SHIFT_ONE_BIT) XOR #mask;
	    ELSE
	      // Shift left without division
	      #tempCRC := SHL(IN := #tempCRC, N := #SHIFT_ONE_BIT);
	    END_IF;
	  END_FOR;
	END_REGION

	REGION Outputs assignment
	  #LGF_CalcCRC8For1Byte := #tempCRC;
	  // no error handling needed
	  ENO := TRUE;
	END_REGION

END_FUNCTION

FUNCTION "LGF_CalcCRC8Advanced" : Byte
{ S7_Optimized_Access := 'TRUE' }
AUTHOR : Siemens_Industry_Support
FAMILY : LGF
NAME : LGF_CRC8Advanced
   VAR_INPUT
      initValue { S7_PredefinedAssignment := '16#00'} : Byte;
      mask { S7_PredefinedAssignment := '16#00'} : Byte;
      finalXorValue { S7_PredefinedAssignment := '16#00'} : Byte;
      reflectInput { S7_PredefinedAssignment := 'FALSE'} : Bool;
      reflectResult { S7_PredefinedAssignment := 'FALSE'} : Bool;
      noOfElements { S7_PredefinedAssignment := '0'} : UInt;
   END_VAR

   VAR_OUTPUT
      error : Bool;
      status : Word;
   END_VAR

   VAR_IN_OUT
      "array" : Array[*] of Byte;
   END_VAR

   VAR_TEMP
      tempInput : Byte;
      tempCRC : Byte;
      tempInvCRC : Byte;
      tempLowerLimit : DInt;
      tempUpperLimit : DInt;
      tempIndexArray : DInt;
      tempIndexCRC : DInt;
   END_VAR

   VAR CONSTANT
      SHIFT_ONE_BIT : UInt := 1;
      ARRAY_FIRST_DIMENSION : UInt := 1;
      CRC_LOOP_LOWER_LIMIT : DInt := 0;
      CRC_LOOP_UPPER_LIMIT : DInt := 7;
      STATUS_NO_ERROR : Word := 16#0000;
      ERR_NO_OF_ELEMENTS : Word := 16#8400;
   END_VAR


BEGIN
	REGION Block info header
	  //===============================================================================
	  // SIEMENS AG / (c)Copyright 2019
	  //-------------------------------------------------------------------------------
	  // Title:            LGF_CRC8Advanced
	  // Comment/Function: This function makes a CRC calculation according
	  //                   to the CRC-8 advanced algorithm
	  //                   advanced because of reflect In/Out and final XOR combination
	  // Library/Family:   LGF (Library General Functions)
	  // Author:           Siemens Digital Industry Support
	  // Tested with:      CPU 1515F-2 PN FW:V2.6
	  // Engineering:      TIA Portal V15.1 Update 2
	  // Restrictions:     ENO disabled - no error handling, no failure possible
	  // Requirements:     PLC (S7-1200 / S7-1500)
	  //-------------------------------------------------------------------------------
	  // Change log table:
	  // Version  | Date       | Expert in charge       | Changes applied
	  //----------|------------|------------------------|------------------------------
	  // 01.00.00 16.12.2019  Simatic Systems Support
	  //                      first release, copied from "LGF_CalcCRC32Advanced"
	  // 03.00.00 23.04.2020  Simatic Systems Support
	  //                      Set version to V3.0.0, harmonize the version of the whole library
	  // 03.00.01 12.11.2020  Simatic Systems Support
	  //                      Insert documentation
	  //                      Assign default start values to optional inputs - `initValue`, `mask`, `finalXorValue`, `reflectInput`, `reflectResult`
	  // 03.01.00 14.04.2023  Simatic Systems Support
	  //                      Add input `noOfElements` to assign length to be converted different from array size
	  //                      Add outputs `error` and `status` display a wrong assignment to `noOfElements`
	  //=============================================================================
	END_REGION Block info header

	REGION DESCRIPTION
	  (/**/)
	END_REGION DESCRIPTION

	REGION Initialization and input data processing
	  // Defining initial value for algorithm
	  #tempCRC := #initValue;
	  // Input array size calculation
	  #tempLowerLimit := LOWER_BOUND(ARR := #array, DIM := #ARRAY_FIRST_DIMENSION);
	  #tempUpperLimit := UPPER_BOUND(ARR := #array, DIM := #ARRAY_FIRST_DIMENSION);

	  // check paramter `noOfELements`, if gretaer than zero check if fits to array size
	  IF #noOfElements > 0 THEN
	    IF #noOfElements > (#tempUpperLimit - #tempLowerLimit + 1) THEN
	      #status := #ERR_NO_OF_ELEMENTS;
	      #error := TRUE;
	      ENO := FALSE;
	      #LGF_CalcCRC8Advanced := #tempCRC;
	      RETURN;
	    ELSE
	      #tempUpperLimit := #tempLowerLimit + #noOfElements - 1;
	    END_IF;
	  END_IF;
	END_REGION

	REGION CRC calculation
	  FOR #tempIndexArray := #tempLowerLimit TO #tempUpperLimit DO

	    IF #reflectInput THEN
	      // Reverse bit order in input byte
	      #tempInput.%X7 := #array[#tempIndexArray].%X0;
	      #tempInput.%X6 := #array[#tempIndexArray].%X1;
	      #tempInput.%X5 := #array[#tempIndexArray].%X2;
	      #tempInput.%X4 := #array[#tempIndexArray].%X3;
	      #tempInput.%X3 := #array[#tempIndexArray].%X4;
	      #tempInput.%X2 := #array[#tempIndexArray].%X5;
	      #tempInput.%X1 := #array[#tempIndexArray].%X6;
	      #tempInput.%X0 := #array[#tempIndexArray].%X7;
	    ELSE
	      #tempInput := #array[#tempIndexArray];
	    END_IF;

	    // Perform division using XOR function for appropriate byte in the array
	    #tempCRC := #tempCRC XOR #tempInput;

	    FOR #tempIndexCRC := #CRC_LOOP_LOWER_LIMIT TO #CRC_LOOP_UPPER_LIMIT DO
	      // Check if MSB is set
	      IF #tempCRC.%X7 THEN
	        // Shift left and perform division by mask polynomial using XOR function
	        #tempCRC := SHL(IN := #tempCRC, N := #SHIFT_ONE_BIT) XOR #mask;
	      ELSE
	        // Shift left without division
	        #tempCRC := SHL(IN := #tempCRC, N := #SHIFT_ONE_BIT);
	      END_IF;
	    END_FOR;

	  END_FOR;
	END_REGION

	REGION Outputs assignment
	  IF #reflectResult THEN
	    // Reverse bit order in CRC checksum
	    #tempInvCRC.%X7 := #tempCRC.%X0;
	    #tempInvCRC.%X6 := #tempCRC.%X1;
	    #tempInvCRC.%X5 := #tempCRC.%X2;
	    #tempInvCRC.%X4 := #tempCRC.%X3;
	    #tempInvCRC.%X3 := #tempCRC.%X4;
	    #tempInvCRC.%X2 := #tempCRC.%X5;
	    #tempInvCRC.%X1 := #tempCRC.%X6;
	    #tempInvCRC.%X0 := #tempCRC.%X7;

	    #LGF_CalcCRC8Advanced := #tempInvCRC XOR #finalXorValue;
	  ELSE
	    #LGF_CalcCRC8Advanced := #tempCRC XOR #finalXorValue;
	  END_IF;

	  #status := #STATUS_NO_ERROR;
	  #error := FALSE;
	  ENO := TRUE;
	END_REGION

END_FUNCTION

FUNCTION "LGF_IsParityEven" : Bool
{ S7_Optimized_Access := 'TRUE' }
AUTHOR : Siemens_SIMATIC_Systems_Support
FAMILY : LGF
NAME : LGF_IsParityEven
   VAR_INPUT
      doubleWord : DWord;
   END_VAR

   VAR_TEMP
      tempDword : DWord;
   END_VAR

   VAR CONSTANT
      SHIFT_ONE_BIT : USInt := 1;
      SHIFT_TWO_BIT : USInt := 2;
      SHIFT_TO_RESULT : USInt := 28;
      MASK_FOR_RESULT : DWord := 16#11111111;
   END_VAR


BEGIN
	REGION Block info header
	  //============================================================================
	  // SIEMENS AG / (c)Copyright 2018
	  //----------------------------------------------------------------------------
	  // Title:            LGF_IsParityEven
	  // Comment/Function: check if parity in input tag is even
	  //                   if number of bits is even, return TRUE
	  //                   https://graphics.stanford.edu/~seander/bithacks.html#ParityMultiply
	  // Library/Family:   LGF (Library General Functions)
	  // Author:           Siemens Digital Industry Support
	  // Tested with:      S7-PLCSIM Advanced V2.0 SP1
	  // Engineering:      TIA Portal V15 Update 2
	  // Restrictions:     ENO not needed, no error possible
	  // Requirements:     PLC (S7-1200 / S7-1500)
	  //-------------------------------------------------------------------------------
	  // Change log table:
	  // Version  | Date       | Expert in charge       | Changes applied
	  //----------|------------|------------------------|------------------------------
	  // 01.00.00 | 2019.11.28 | Simatic Systems Support
	  //                         First released version
	  // 03.00.00 | 23.04.2020 | Simatic Systems Support | Set version to V3.0.0
	  //                         harmonize the version of the whole library
	  // 03.00.01 | 12.11.2020 | Simatic Systems Support
	  //                         Insert documentation
	  //=============================================================================
	END_REGION Block info header

	REGION DESCRIPTION
	  (/**/)
	END_REGION DESCRIPTION

	REGION Logic
	  #tempDword := #doubleWord; // 32-bit word
	  #tempDword := #tempDword XOR SHR(IN := #tempDword, N := #SHIFT_ONE_BIT);
	  #tempDword := #tempDword XOR SHR(IN := #tempDword, N := #SHIFT_TWO_BIT);
	  #tempDword := UDINT_TO_DWORD(DWORD_TO_UDINT(#tempDword AND #MASK_FOR_RESULT) * DWORD_TO_UDINT(#MASK_FOR_RESULT));

	  #tempDword := SHR(IN := #tempDword, N := #SHIFT_TO_RESULT);

	  // result is stored in LSB
	  #LGF_IsParityEven := NOT #tempDword.%X0;

	  // ENO not needed, no error possible
	  ENO := FALSE;
	END_REGION

END_FUNCTION

FUNCTION_BLOCK "LGF_ShiftRegister"
{ S7_Optimized_Access := 'TRUE' }
AUTHOR : Siemens_Digital_Industry_Support
FAMILY : LGF
NAME : LGF_ShiftRegister
   VAR_INPUT
      shiftLeft : Bool;
      shiftRight : Bool;
      shiftRange { S7_PredefinedAssignment := '1'; S7_HiddenAssignment := 'HideIfNoParamAssigned'} : UInt := 1;
      clear : Bool;
      fill : Bool;
      initialItem { S7_PredefinedAssignment := 'NULL'} : Variant;
   END_VAR

   VAR_OUTPUT
      error { ExternalWritable := 'False'} : Bool;
      status { ExternalWritable := 'False'} : Word;
      subFunctionStatus { ExternalWritable := 'False'} : Word;
   END_VAR

   VAR_IN_OUT
      bufferRegister : Variant;
   END_VAR

   VAR
      statEdgesMem { ExternalAccessible := 'False'; ExternalVisible := 'False'; ExternalWritable := 'False'} : Struct
         shiftCommand { ExternalAccessible := 'False'; ExternalVisible := 'False'; ExternalWritable := 'False'} : Bool;
         clear { ExternalAccessible := 'False'; ExternalVisible := 'False'; ExternalWritable := 'False'} : Bool;
      END_STRUCT;
   END_VAR

   VAR_TEMP
      tempEdges : Struct
         shiftLeft : Bool;
         shiftRight : Bool;
         clear : Bool;
      END_STRUCT;
      tempInternalError : Int;
      tempBufferSize : UDInt;
      tempCounter : Int;
   END_VAR

   VAR CONSTANT
      NO_INTERNAL_ERROR : Int := 16#0000;
      INDEX_BEGINNING : Int := 0;
      ONE_ELEMENT : UDInt := 1;
      BUFFER_SIZE_CORRECTION : UDInt := 1;
      STATUS_NO_ERROR : Word := 16#0000;
      STATUS_NO_CURRENT_JOBS : Word := 16#7000;
      ERR_NO_ARRAY : Word := 16#8200;
      ERR_CLEARING_WITHOUT_INITIAL_ITEM : Word := 16#8201;
      ERR_FILL_WITHOUT_INITIAL_ITEM : Word := 16#8202;
      ERR_WRONG_TYPE_INITIAL_ITEM : Word := 16#8203;
      ERR_MORE_THAN_ONE_COMMAND : Word := 16#8401;
      ERR_IN_SHIFT_RANGE : Word := 16#8402;
      ERR_CLEAR_BUFFER : Word := 16#8610;
      ERR_SHIFT_BUFFER_LEFT : Word := 16#8611;
      ERR_SHIFT_BUFFER_LEFT_FILL : Word := 16#8612;
      ERR_SHIFT_BUFFER_RIGHT : Word := 16#8622;
      ERR_SHIFT_BUFFER_RIGHT_FILL : Word := 16#8622;
   END_VAR


BEGIN
	REGION Block info header
	  //===============================================================================
	  // SIEMENS AG / (c)Copyright 2019
	  //-------------------------------------------------------------------------------
	  // Title:            LGF_ShiftRegister
	  // Comment/Function: The Function represnts a shift register for any kind of Datatype (using `variant`) - it can be used as a kind of a ring buffer.
	  //                   It is possible to shift the register array left (index `array[n]:=array[n+1]`) or right (index a`array[n]:=array[n-1]`).
	  //                   As this is a real shift operation, it may causes some runtime effects while using big array sizes to move.
	  //                   It could be used for pusing the material traking UDT trouf the maschin, e.g. a rotary indexing table
	  //                   Please consider that a FIFO  or LIFO storage, based on indexes, could be used as well for most applications.
	  // Library/Family:   LGF (Library General Functions)
	  // Author:           Siemens Digital Industry Support
	  // Tested with:      CPU 1515F-2 PN FW:V2.6
	  // Engineering:      TIA Portal V16 Update 4
	  // Restrictions:     ENO disabled - error handling done with error and status
	  // Requirements:     PLC (S7-1200 / S7-1500)
	  //-------------------------------------------------------------------------------
	  // Change log table:
	  // Version  | Date       | Expert in charge       | Changes applied
	  //----------|------------|------------------------|------------------------------
	  // 01.00.00 03.07.2018  Siemens Industry Online Support
	  //                      First released version
	  // 03.00.00 09.04.2021  Simatic Systems Support
	  //                      Refactoring and alignment to Datatype Variant
	  //                      Insert documentation
	  //=============================================================================
	END_REGION Block info header

	REGION DESCRIPTION
	  (/**/)
	END_REGION DESCRIPTION

	REGION Block execution control
	  // Collect edges
	  #tempEdges.shiftLeft := #shiftLeft AND NOT #statEdgesMem.shiftCommand;
	  #tempEdges.shiftRight := #shiftRight AND NOT #statEdgesMem.shiftCommand;
	  #tempEdges.clear := #clear AND NOT #statEdgesMem.clear;
	  // Store values for edge detection
	  #statEdgesMem.shiftCommand := #shiftLeft OR #shiftRight;
	  #statEdgesMem.clear := #clear;

	  // This program code section is only executed if no trigger input is active
	  IF NOT (#shiftLeft OR #shiftRight OR #clear) THEN
	    // If an error occurred during program execution,
	    // the status "No Current Job" is used 16#7000 afterwarts when the triggers are reseted
	    #error := FALSE;
	    #status := #STATUS_NO_CURRENT_JOBS;
	    #subFunctionStatus := #STATUS_NO_ERROR;
	    RETURN;

	  ELSIF ((BOOL_TO_USINT(#shiftLeft) + BOOL_TO_USINT(#shiftRight) + BOOL_TO_USINT(#clear)) > 1) THEN
	    #error := TRUE;
	    #status := #ERR_MORE_THAN_ONE_COMMAND;
	    #subFunctionStatus := #STATUS_NO_ERROR;
	    RETURN;
	  END_IF;
	END_REGION Block execution control

	REGION Validation of inputs
	  // Check whether the ring #buffer is an ARRAY.
	  // IF so, the number OF the ARRAY elements is read out.
	  // IF it is NOT an ARRAY, the program execution is terminated at this point
	  IF IS_ARRAY(#bufferRegister) THEN
	    #tempBufferSize := CountOfElements(#bufferRegister);
	  ELSE
	    #error := TRUE;
	    #status := #ERR_NO_ARRAY;
	    #subFunctionStatus := #STATUS_NO_ERROR;
	    RETURN;
	  END_IF;

	  // Check if number of movements is in a plausible and valid range
	  // -> Has to be lees than the buffer size
	  IF #shiftRange >= #tempBufferSize THEN
	    #error := TRUE;
	    #status := #ERR_IN_SHIFT_RANGE;
	    #subFunctionStatus := #STATUS_NO_ERROR;
	    RETURN;
	  END_IF;

	  // If clearBuffer has rising edge, the buffer is initialized by initial values
	  // Check whether the initial value OF the ring #buffer
	  // matches the entry (tag #item). IF the data types DO NOT match,
	  // the program execution is terminated at this point
	  IF (#tempEdges.clear AND #initialItem = NULL) THEN
	    #error := TRUE;
	    #status := #ERR_CLEARING_WITHOUT_INITIAL_ITEM;
	    #subFunctionStatus := #STATUS_NO_ERROR;
	    RETURN;

	    // If Fill is activatet, an inital item has to be presnt
	  ELSIF (#fill AND #initialItem = NULL) THEN
	    #error := TRUE;
	    #status := #ERR_FILL_WITHOUT_INITIAL_ITEM;
	    #subFunctionStatus := #STATUS_NO_ERROR;
	    RETURN;

	    // If clearing or filling is selected, the input types must match
	  ELSIF ((#tempEdges.clear OR #fill) AND #initialItem <> NULL)
	    AND (TypeOfElements(#bufferRegister) <> TypeOf(#initialItem))
	  THEN
	    #error := TRUE;
	    #status := #ERR_WRONG_TYPE_INITIAL_ITEM;
	    #subFunctionStatus := #STATUS_NO_ERROR;
	    RETURN;
	  END_IF;
	END_REGION Validation of inputs

	REGION Clear Buffer
	  // If clearBuffer has rising edge, the buffer is initialized by initial values
	  IF #tempEdges.clear THEN
	    // Run through buffer and overwrite all elements with its initial item element
	    FOR #tempCounter := #INDEX_BEGINNING TO UDINT_TO_INT(#tempBufferSize - #BUFFER_SIZE_CORRECTION) DO
	      #tempInternalError := MOVE_BLK_VARIANT(SRC := #initialItem,
	                                             COUNT := #ONE_ELEMENT,
	                                             SRC_INDEX := #INDEX_BEGINNING,
	                                             DEST_INDEX := #tempCounter,
	                                             DEST => #bufferRegister);
	    END_FOR;

	    // Check whether a local error has occurred.
	    IF (#tempInternalError <> #NO_INTERNAL_ERROR) THEN
	      #error := TRUE;
	      #status := #ERR_CLEAR_BUFFER;
	      #subFunctionStatus := INT_TO_WORD(#tempInternalError);
	      RETURN;
	    END_IF;
	  END_IF;
	END_REGION Clear Buffer

	REGION Shift register algorithm
	  REGION Shift left
	    IF #tempEdges.shiftLeft THEN
	      // Shift whole array elemnts from N --> N-1
	      #tempInternalError :=
	      MOVE_BLK_VARIANT(SRC := #bufferRegister,
	                       COUNT := #tempBufferSize - #shiftRange,
	                       SRC_INDEX := #shiftRange,
	                       DEST_INDEX := 0,
	                       DEST => #bufferRegister);

	      // Check whether a local error has occurred
	      IF (#tempInternalError <> #NO_INTERNAL_ERROR) THEN
	        #error := TRUE;
	        #status := #ERR_SHIFT_BUFFER_LEFT;
	        #subFunctionStatus := INT_TO_WORD(#tempInternalError);
	        RETURN;
	      END_IF;

	      REGION Fill after shift left
	        IF #fill THEN
	          // Run through buffer and overwrite all elements with its initial item element
	          FOR #tempCounter := UINT_TO_INT(#shiftRange) TO UDINT_TO_INT(#tempBufferSize - #BUFFER_SIZE_CORRECTION) DO
	            // Overwrite the "old" values after shift
	            #tempInternalError := MOVE_BLK_VARIANT(SRC := #initialItem,
	                                                   COUNT := #ONE_ELEMENT,
	                                                   SRC_INDEX := #INDEX_BEGINNING,
	                                                   DEST_INDEX := #tempCounter,
	                                                   DEST => #bufferRegister);

	            // Check whether a local error has occurred
	            IF (#tempInternalError <> #NO_INTERNAL_ERROR) THEN
	              #error := TRUE;
	              #status := #ERR_SHIFT_BUFFER_LEFT_FILL;
	              #subFunctionStatus := INT_TO_WORD(#tempInternalError);
	              RETURN;
	            END_IF;
	          END_FOR;
	        END_IF;
	      END_REGION Fill after shift left
	    END_IF;
	  END_REGION Shift left

	  REGION Shift right
	    IF #tempEdges.shiftRight THEN
	      // Shift whole array elemnsts from N --> N+1
	      #tempInternalError := MOVE_BLK_VARIANT(SRC := #bufferRegister,
	                                             COUNT := #tempBufferSize - #shiftRange,
	                                             SRC_INDEX := 0,
	                                             DEST_INDEX := #shiftRange,
	                                             DEST => #bufferRegister);

	      // Check whether a local error has occurred
	      IF (#tempInternalError <> #NO_INTERNAL_ERROR) THEN
	        #error := TRUE;
	        #status := #ERR_SHIFT_BUFFER_RIGHT;
	        #subFunctionStatus := INT_TO_WORD(#tempInternalError);
	        RETURN;
	      END_IF;

	      REGION Fill after shift right
	        IF #fill THEN
	          // Run through buffer and overwrite all elements with its initial item element
	          FOR #tempCounter := #INDEX_BEGINNING TO UDINT_TO_INT(#shiftRange - #BUFFER_SIZE_CORRECTION) DO
	            // Overwrite the "old" values after shift
	            #tempInternalError := MOVE_BLK_VARIANT(SRC := #initialItem,
	                                                   COUNT := #ONE_ELEMENT,
	                                                   SRC_INDEX := #INDEX_BEGINNING,
	                                                   DEST_INDEX := #tempCounter,
	                                                   DEST => #bufferRegister);

	            // Check whether a local error has occurred
	            IF (#tempInternalError <> #NO_INTERNAL_ERROR) THEN
	              #error := TRUE;
	              #status := #ERR_SHIFT_BUFFER_LEFT_FILL;
	              #subFunctionStatus := INT_TO_WORD(#tempInternalError);
	              RETURN;
	            END_IF;
	          END_FOR;
	        END_IF;
	      END_REGION Fill after shift right
	    END_IF;
	  END_REGION Shift right
	END_REGION Shift register algorithm

	REGION Writing to outputs
	  #error := FALSE;
	  #status := #STATUS_NO_ERROR;
	  #subFunctionStatus := #STATUS_NO_ERROR;
	  // No error handling by ENO needed
	  ENO := TRUE;
	END_REGION Writing to outputs

END_FUNCTION_BLOCK

